ABB RAPID module: SinglePartTemplate.mod

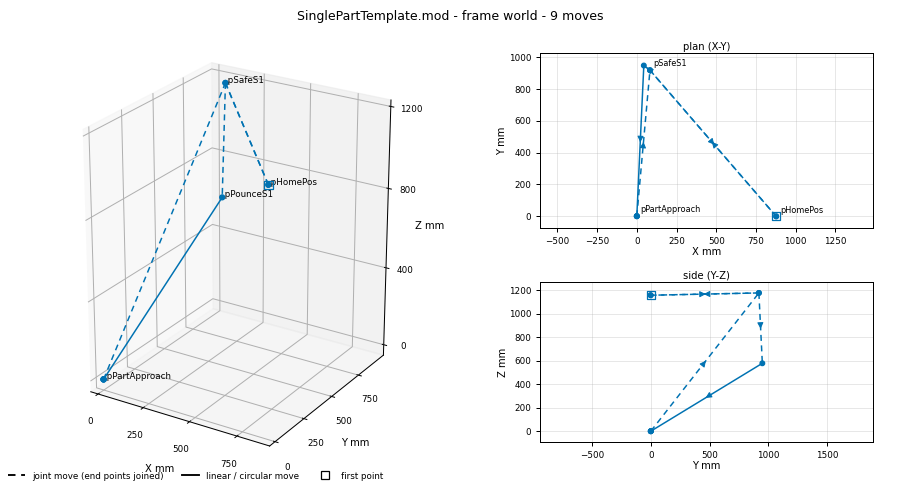
[picture p0: tool path of SinglePartTemplate.mod in frame world, 9 of 9 moves have a stored position in this frame; points joined in program order, loops and branches not executed]
MODULE SinglePartTemplate
  ! ------------------------------------------------------------------
  ! Single-part welding template
  !
  ! Purpose:
  !   - Run one part only (no multi-part branching)
  !   - Keep nozzle cleaning and BullsEye tool check available
  !   - Provide a copy/paste starting point for new part files
  !
  ! Dependencies:
  !   - LogicZ (home/safe/pounce positions + rTC2013)
  !   - BE_User1 (BECheckToolb for BullsEye)
  !   - mTSC (optional torch cleaner if you prefer MechCleanGun)
  ! ------------------------------------------------------------------

  LOCAL PERS bool bUseTorchClean := TRUE;
  LOCAL PERS bool bUseBullseye := TRUE;

  ! Placeholder weld/seam data for the template. Replace with real values.
  LOCAL PERS welddata weldPart := [0,0,[1,0,0,0,0,0,0,0,0],[0,0,0,0,0,0,0,0,0]];
  LOCAL PERS seamdata seamPart := [1,1,[1,0,0,0,0,0,0,0,0],0,0,0,0,0,[0,0,0,0,0,0,0,0,0],0,0,[0,0,0,0,0,0,0,0,0],0,0,[0,0,0,0,0,0,0,0,0],0];

  ! Placeholder targets for the weld path. Replace with taught points.
  LOCAL CONST robtarget pPartApproach := [[0,0,0],[1,0,0,0],[0,0,0,0],[9E+09,9E+09,9E+09,9E+09,9E+09,9E+09]];
  CONST robtarget pPartStart := [[0,0,0],[1,0,0,0],[0,0,0,0],[9E+09,9E+09,9E+09,9E+09,9E+09,9E+09]];
  CONST robtarget pPartEnd := [[0,0,0],[1,0,0,0],[0,0,0,0],[9E+09,9E+09,9E+09,9E+09,9E+09,9E+09]];
  CONST robtarget pPartDepart := [[0,0,0],[1,0,0,0],[0,0,0,0],[9E+09,9E+09,9E+09,9E+09,9E+09,9E+09]];

  PROC RunSinglePartTemplate()
    TPWrite "Single-part template start";

    ! Optional BullsEye tool check before running a part.
    IF bUseBullseye THEN
      BECheckToolb;
    ENDIF

    ! Optional nozzle cleaning/reaming before the part weld.
    IF bUseTorchClean THEN
      rTC2013;
      ! Alternative: MechCleanGun;  ! From mTSC.mod
    ENDIF

    MoveJ pHomePos, v800, fine, tWeldGun;
    MoveJ pSafeS1, v800, fine, tWeldGun;
    MoveJ pPounceS1, v800, fine, tWeldGun;

    ! ----------------------------------------------------------------
    ! Single-part weld path (edit only the weld start/end points).
    ! ----------------------------------------------------------------
    MoveL pPartApproach, v200, z10, tWeldGun;
    ArcLStart pPartStart, v30, seamPart, weldPart, fine, tWeldGun;
    ArcLEnd pPartEnd, v30, seamPart, weldPart, fine, tWeldGun;
    MoveL pPartDepart, v200, z10, tWeldGun;

    MoveJ pSafeS1, v800, fine, tWeldGun;
    MoveJ pHomePos, v800, fine, tWeldGun;

    TPWrite "Single-part template complete";
  ENDPROC
ENDMODULE
